// TIA Portal V18 export
FUNCTION "fcMain" : Void   // FC2, LAD
// stored: Access Published, Namespace nsMainPerceuse, SetENOAutomatically false
   VAR_INPUT
      iStart : Bool;
      iFaster : Bool;
      iSlower : Bool;
   END_VAR
   VAR_OUTPUT
      oStatus : Bool;
   END_VAR
   VAR_IN_OUT
      ioSpeed : UDInt;
   END_VAR
BEGIN

REGION Network 1
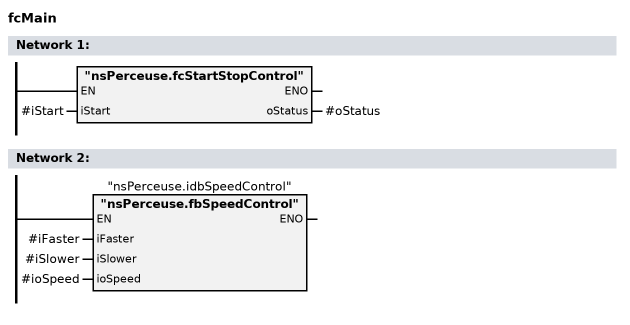
   RUNG wire#powerrail
      "nsPerceuse.fcStartStopControl"(iStart := #iStart, oStatus => #oStatus)
   END_RUNG
   // the same network as SCL:
   "nsPerceuse.fcStartStopControl"(iStart := #iStart, oStatus => #oStatus);
END_REGION

REGION Network 2
   RUNG wire#powerrail
      "nsPerceuse.idbSpeedControl"(iFaster := #iFaster, iSlower := #iSlower, ioSpeed := #ioSpeed)
   END_RUNG
   // the same network as SCL:
   "nsPerceuse.idbSpeedControl"(iFaster := #iFaster, iSlower := #iSlower, ioSpeed := #ioSpeed);   // "nsPerceuse.fbSpeedControl"
END_REGION
END_FUNCTION
